INTERFACE ValueRead EXTENDS ValueWithType

METHOD Get
VAR_INPUT
	destination : ANY;
END_VAR
END_METHOD

METHOD GetAsString : T_MaxString
VAR_INPUT
END_VAR
END_METHOD

METHOD GetAsType
VAR_INPUT
	destination : __SYSTEM.AnyType;
END_VAR
END_METHOD

END_INTERFACE

(* stored: Version 1.1.0.1, ProductVersion 3.1.4024.15
   Itf ValueRead: Id {a1041c65-021b-4dce-8116-28824fba3b5b}
   Method Get: Id {bcbdc575-c1a9-4b54-b3d9-1957ab36cce4}
   Method GetAsString: Id {db6ccb01-b500-4d35-814b-f9adb612e8b7}
   Method GetAsType: Id {34d57f9b-0840-4c34-a336-e72acbc66aa9} *)
